FUNCTION MotorController : BOOl
VAR_INPUT
	iMotor1 : I_Motor;
	bRun : BOOL;
	fSpeed : REAL;
END_VAR
VAR
END_VAR


IF bRun THEN
	iMotor1.Start();
ELSE
	iMotor1.Stop();
END_IF

END_FUNCTION

(* stored: Version 1.1.0.1, ProductVersion 3.1.4024.16
   POU MotorController: Id {ef45ef2d-b6ed-4d33-bf44-a2461ae43f9a}, SpecialFunc None *)
